// SIMATIC S7-200 project (STEP 7-Micro/WIN), CPU 226 REL 02.00

ORGANIZATION_BLOCK OB_1:OB1
TITLE=PROGRAM COMMENTS
BEGIN
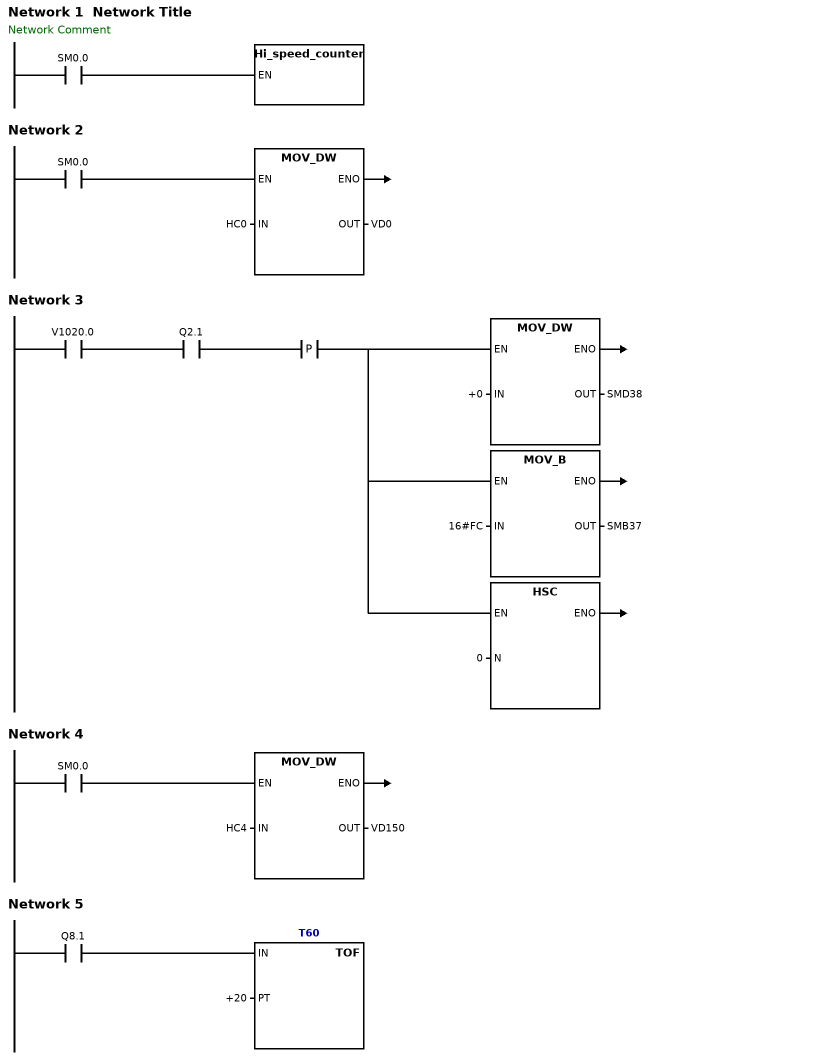
Network 1 // Network Title
// Network Comment
LD     SM0.0
CALL   Hi_speed_counter:SBR1
Network 2
LD     SM0.0
MOVD   HC0, VD0
Network 3
LD     V1020.0
A      Q2.1
EU
MOVD   +0, SMD38
MOVB   16#FC, SMB37
HSC    0
Network 4
LD     SM0.0
MOVD   HC4, VD150
Network 5
LD     Q8.1
TOF    T60, +20
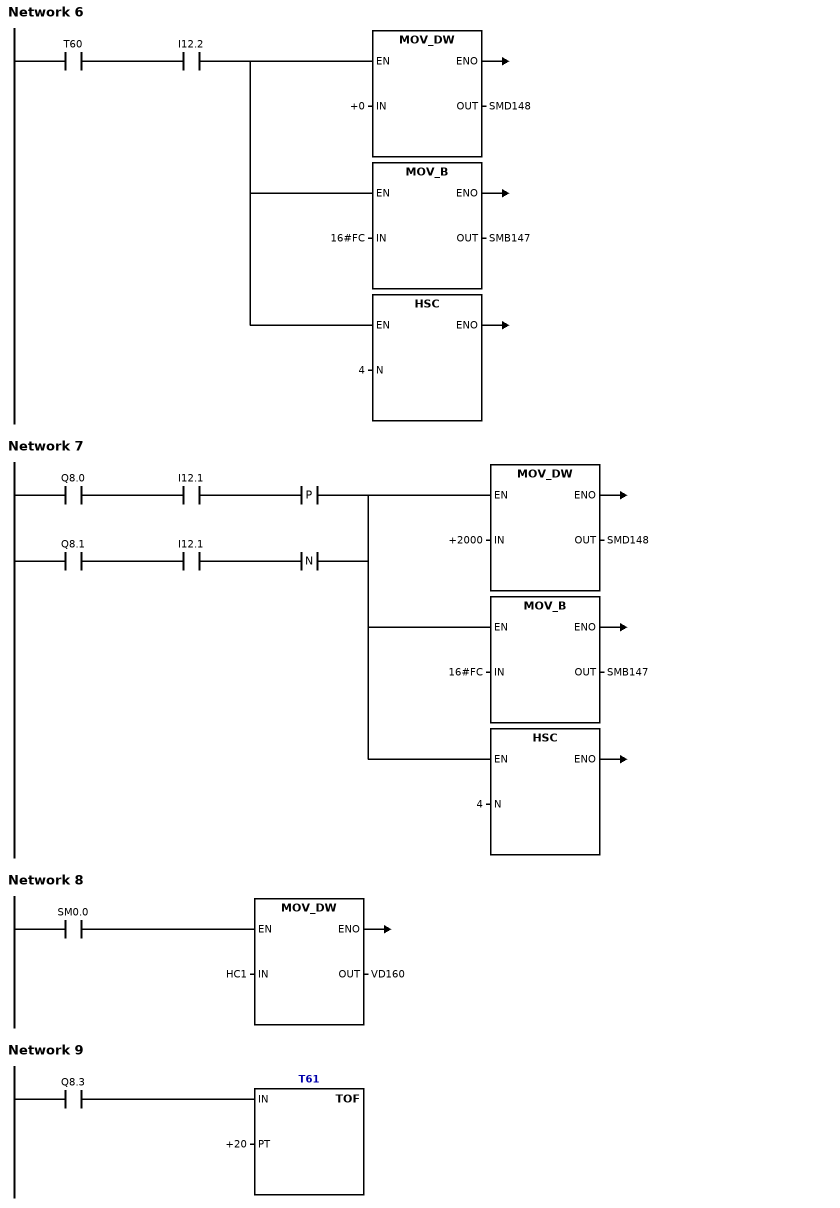
Network 6
LD     T60
A      I12.2
MOVD   +0, SMD148
MOVB   16#FC, SMB147
HSC    4
Network 7
LD     Q8.0
A      I12.1
EU
LD     Q8.1
A      I12.1
ED
OLD
MOVD   +2000, SMD148
MOVB   16#FC, SMB147
HSC    4
Network 8
LD     SM0.0
MOVD   HC1, VD160
Network 9
LD     Q8.3
TOF    T61, +20
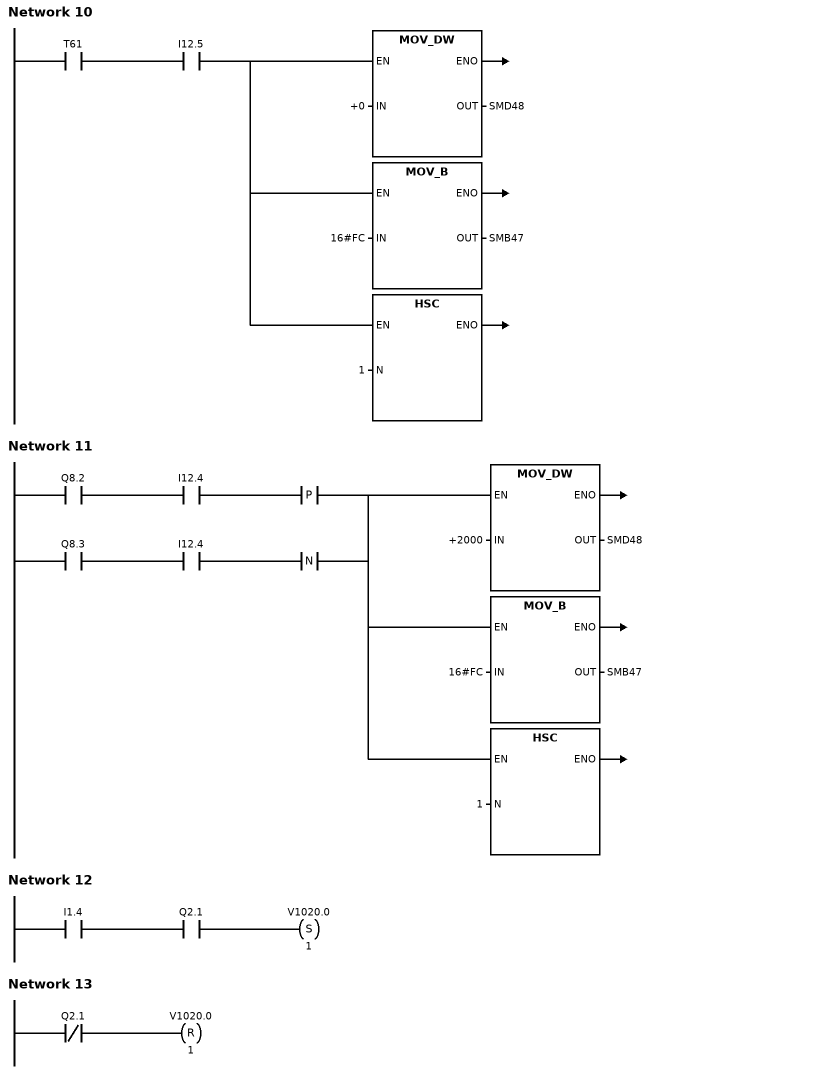
Network 10
LD     T61
A      I12.5
MOVD   +0, SMD48
MOVB   16#FC, SMB47
HSC    1
Network 11
LD     Q8.2
A      I12.4
EU
LD     Q8.3
A      I12.4
ED
OLD
MOVD   +2000, SMD48
MOVB   16#FC, SMB47
HSC    1
Network 12
LD     I1.4
A      Q2.1
S      V1020.0, 1
Network 13
LDN    Q2.1
R      V1020.0, 1
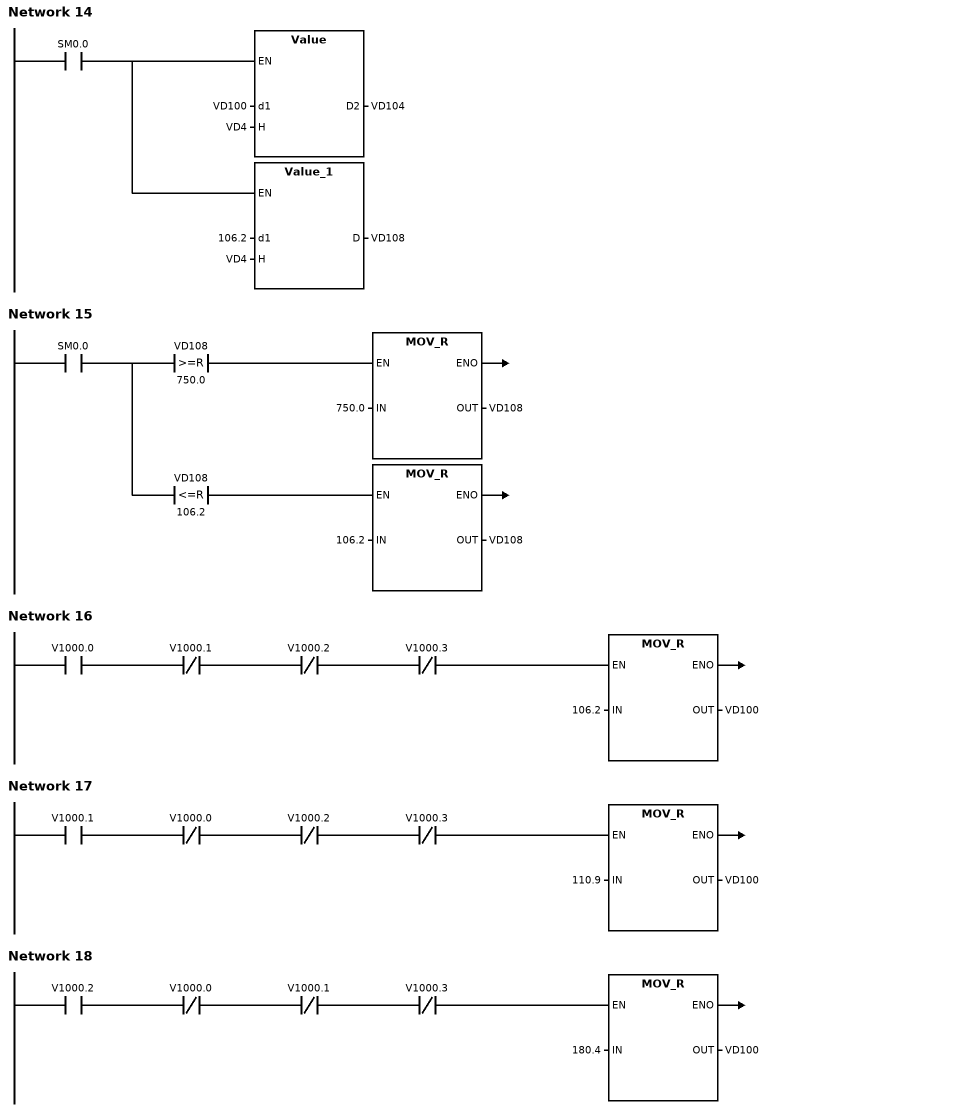
Network 14
LD     SM0.0
CALL   Value:SBR0, VD100, VD4, VD104
CALL   Value_1:SBR10, 106.2, VD4, VD108
Network 15
LD     SM0.0
LPS
AR>=   VD108, 750.0
MOVR   750.0, VD108
LPP
AR<=   VD108, 106.2
MOVR   106.2, VD108
Network 16
LD     V1000.0
AN     V1000.1
AN     V1000.2
AN     V1000.3
MOVR   106.2, VD100
Network 17
LD     V1000.1
AN     V1000.0
AN     V1000.2
AN     V1000.3
MOVR   110.9, VD100
Network 18
LD     V1000.2
AN     V1000.0
AN     V1000.1
AN     V1000.3
MOVR   180.4, VD100
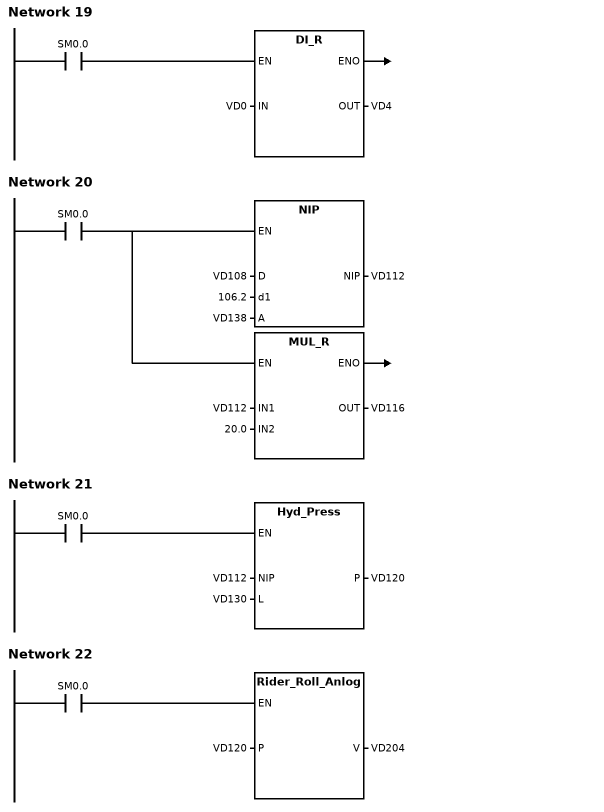
Network 19
LD     SM0.0
DTR    VD0, VD4
Network 20
LD     SM0.0
CALL   NIP:SBR2, VD108, 106.2, VD138, VD112
MOVR   VD112, VD116
*R     20.0, VD116
Network 21
LD     SM0.0
CALL   Hyd_Press:SBR3, VD112, VD130, VD120
Network 22
LD     SM0.0
CALL   Rider_Roll_Anlog:SBR4, VD120, VD204
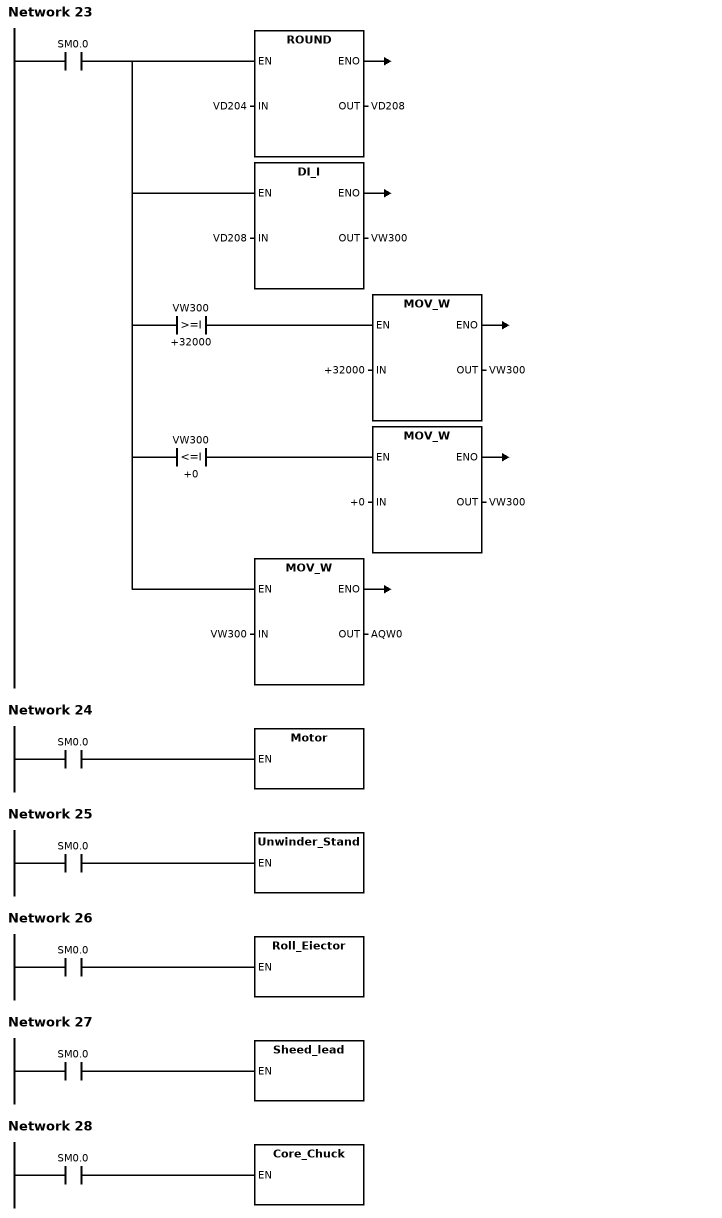
Network 23
LD     SM0.0
LPS
ROUND  VD204, VD208
DTI    VD208, VW300
AW>=   VW300, +32000
MOVW   +32000, VW300
LRD
AW<=   VW300, +0
MOVW   +0, VW300
LPP
MOVW   VW300, AQW0
Network 24
LD     SM0.0
CALL   Motor:SBR5
Network 25
LD     SM0.0
CALL   Unwinder_Stand:SBR6
Network 26
LD     SM0.0
CALL   Roll_Eiector:SBR7
Network 27
LD     SM0.0
CALL   Sheed_lead:SBR8
Network 28
LD     SM0.0
CALL   Core_Chuck:SBR9
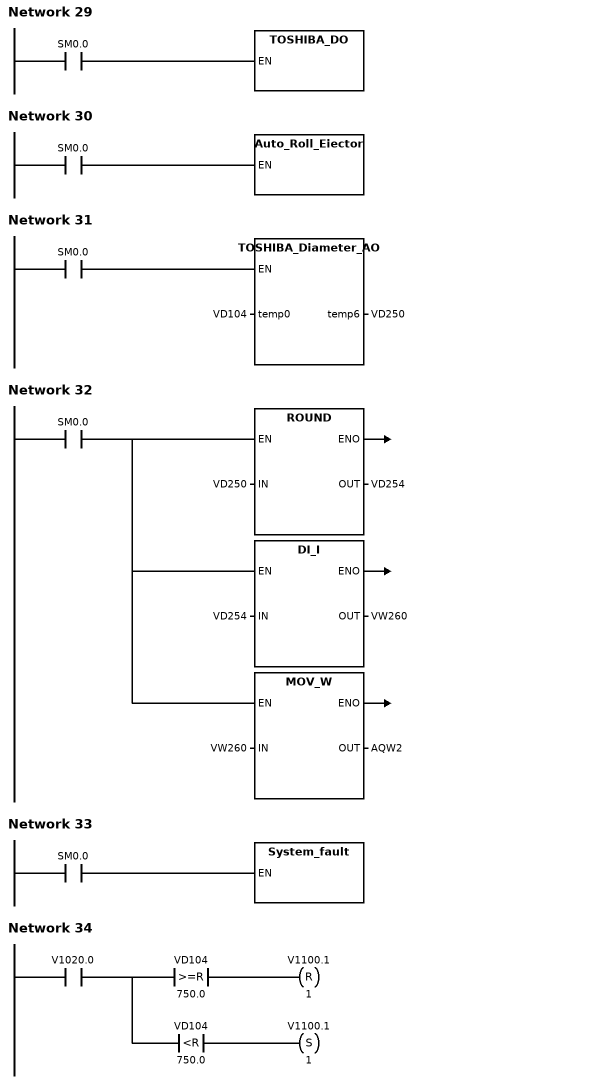
Network 29
LD     SM0.0
CALL   TOSHIBA_DO:SBR11
Network 30
LD     SM0.0
CALL   Auto_Roll_Eiector:SBR12
Network 31
LD     SM0.0
CALL   TOSHIBA_Diameter_AO:SBR13, VD104, VD250
Network 32
LD     SM0.0
ROUND  VD250, VD254
DTI    VD254, VW260
MOVW   VW260, AQW2
Network 33
LD     SM0.0
CALL   System_fault:SBR14
Network 34
LD     V1020.0
LPS
AR>=   VD104, 750.0
R      V1100.1, 1
LPP
AR<    VD104, 750.0
S      V1100.1, 1
END_ORGANIZATION_BLOCK

SUBROUTINE_BLOCK Value:SBR0
TITLE=SUBROUTINE COMMENTS
VAR_INPUT
d1:REAL;	// LD0 
H:REAL;	// LD4 
END_VAR
VAR_OUTPUT
D2:REAL;	// LD8 
END_VAR
BEGIN
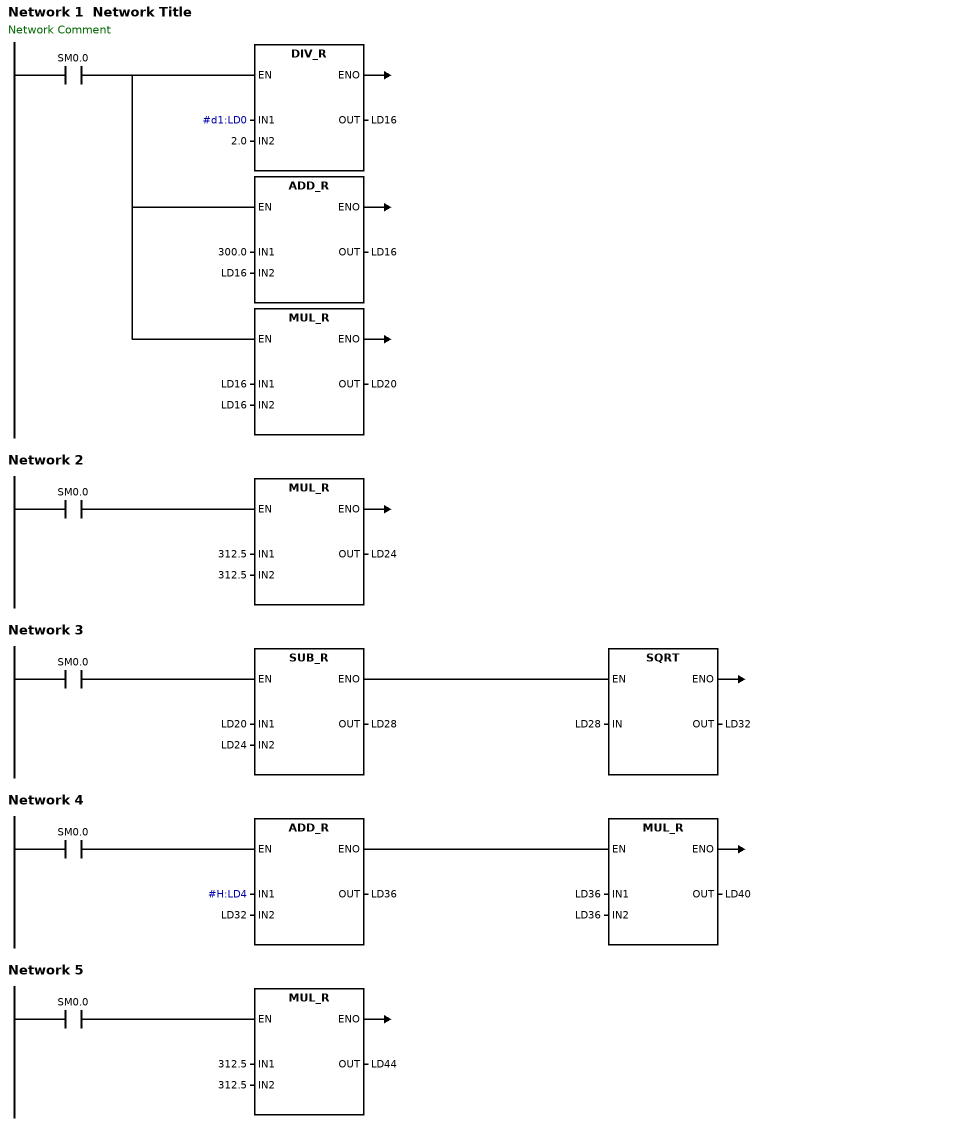
Network 1 // Network Title
// Network Comment
LD     SM0.0
MOVR   #d1:LD0, LD16
/R     2.0, LD16
+R     300.0, LD16
MOVR   LD16, LD20
*R     LD16, LD20
Network 2
LD     SM0.0
MOVR   312.5, LD24
*R     312.5, LD24
Network 3
LD     SM0.0
MOVR   LD20, LD28
AENO
-R     LD24, LD28
AENO
SQRT   LD28, LD32
Network 4
LD     SM0.0
MOVR   #H:LD4, LD36
AENO
+R     LD32, LD36
AENO
MOVR   LD36, LD40
*R     LD36, LD40
Network 5
LD     SM0.0
MOVR   312.5, LD44
*R     312.5, LD44
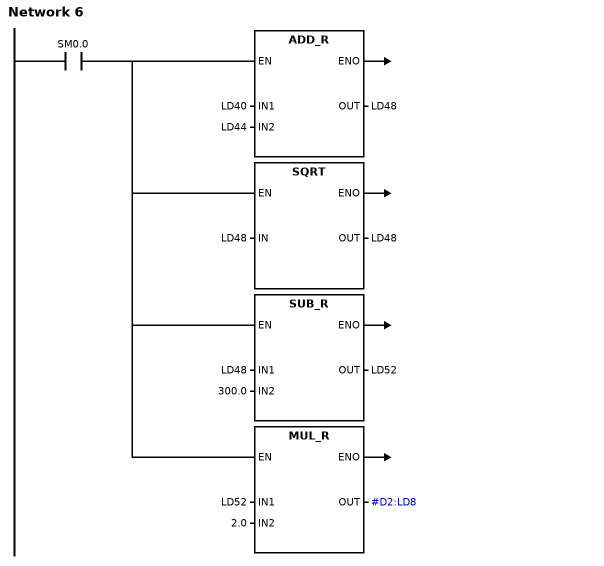
Network 6
LD     SM0.0
MOVR   LD40, LD48
+R     LD44, LD48
SQRT   LD48, LD48
MOVR   LD48, LD52
-R     300.0, LD52
MOVR   LD52, #D2:LD8
*R     2.0, #D2:LD8
END_SUBROUTINE_BLOCK

SUBROUTINE_BLOCK Hi_speed_counter:SBR1
TITLE=
BEGIN
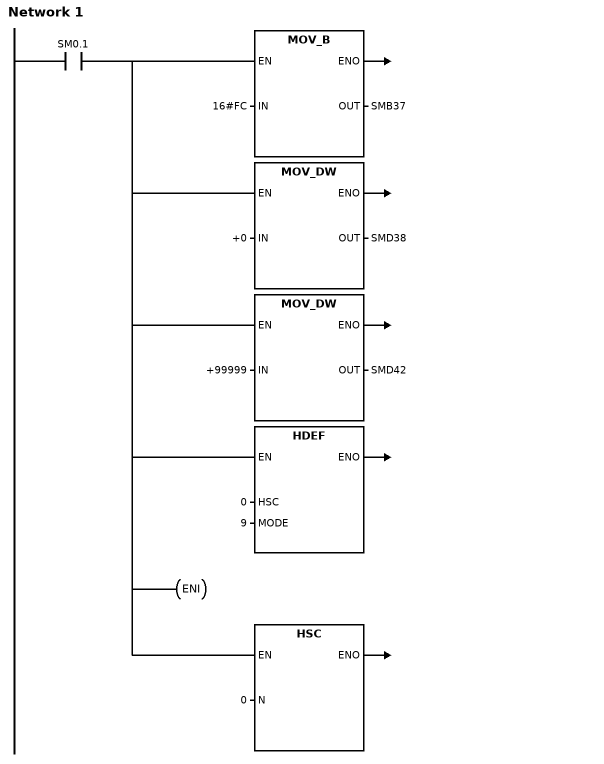
Network 1
LD     SM0.1
MOVB   16#FC, SMB37
MOVD   +0, SMD38
MOVD   +99999, SMD42
HDEF   0, 9
ENI
HSC    0
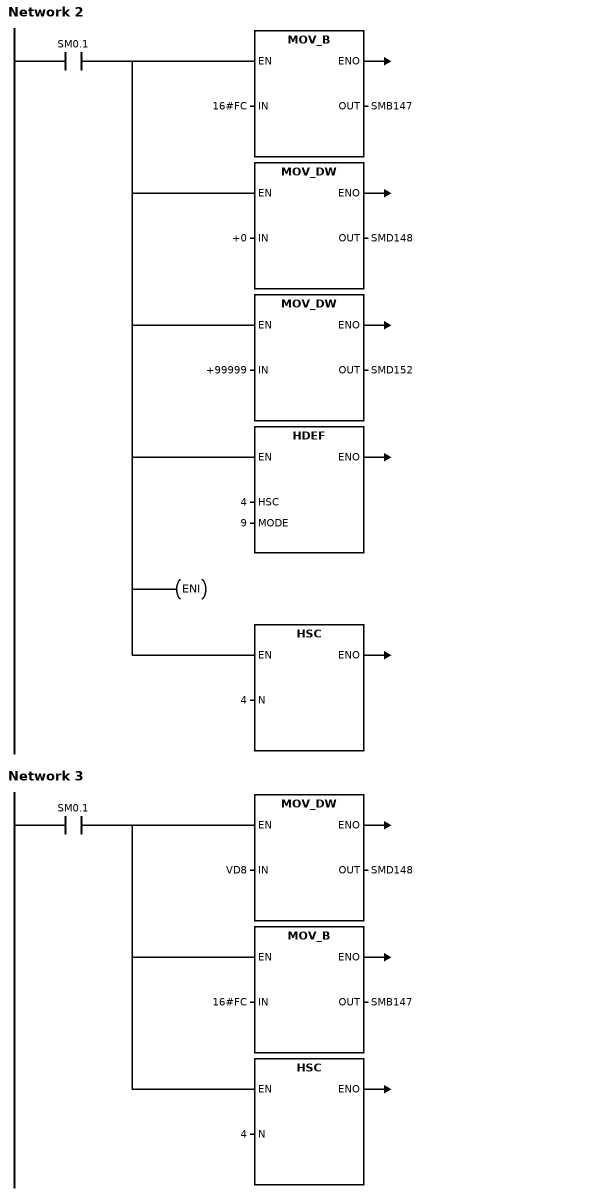
Network 2
LD     SM0.1
MOVB   16#FC, SMB147
MOVD   +0, SMD148
MOVD   +99999, SMD152
HDEF   4, 9
ENI
HSC    4
Network 3
LD     SM0.1
MOVD   VD8, SMD148
MOVB   16#FC, SMB147
HSC    4
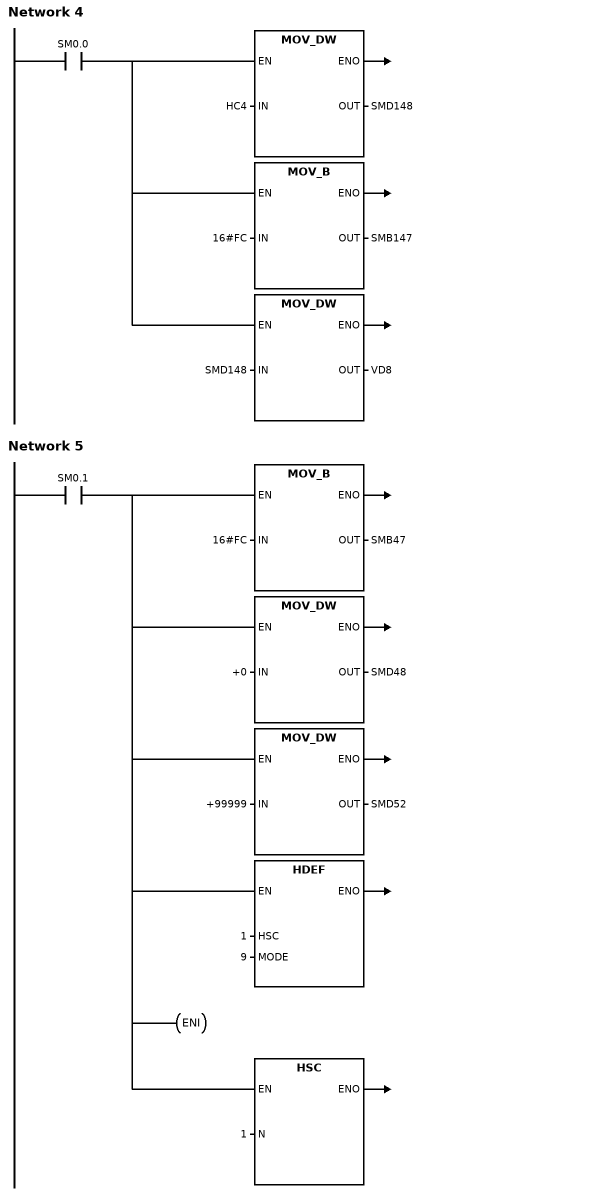
Network 4
LD     SM0.0
MOVD   HC4, SMD148
MOVB   16#FC, SMB147
MOVD   SMD148, VD8
Network 5
LD     SM0.1
MOVB   16#FC, SMB47
MOVD   +0, SMD48
MOVD   +99999, SMD52
HDEF   1, 9
ENI
HSC    1
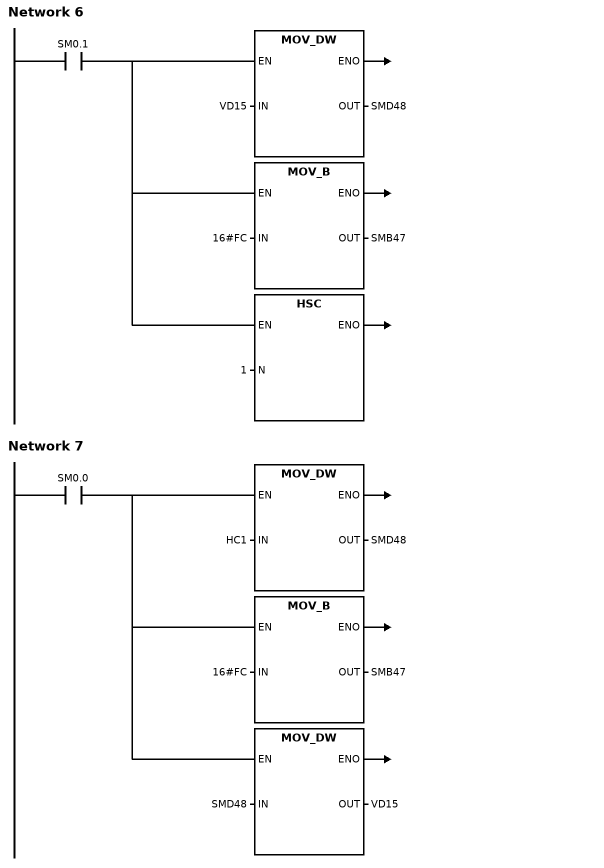
Network 6
LD     SM0.1
MOVD   VD15, SMD48
MOVB   16#FC, SMB47
HSC    1
Network 7
LD     SM0.0
MOVD   HC1, SMD48
MOVB   16#FC, SMB47
MOVD   SMD48, VD15
END_SUBROUTINE_BLOCK

SUBROUTINE_BLOCK NIP:SBR2
TITLE=
VAR_INPUT
D:REAL;	// LD0 
d1:REAL;	// LD4 
A:REAL;	// LD8 
END_VAR
VAR_OUTPUT
NIP:REAL;	// LD12 
END_VAR
BEGIN
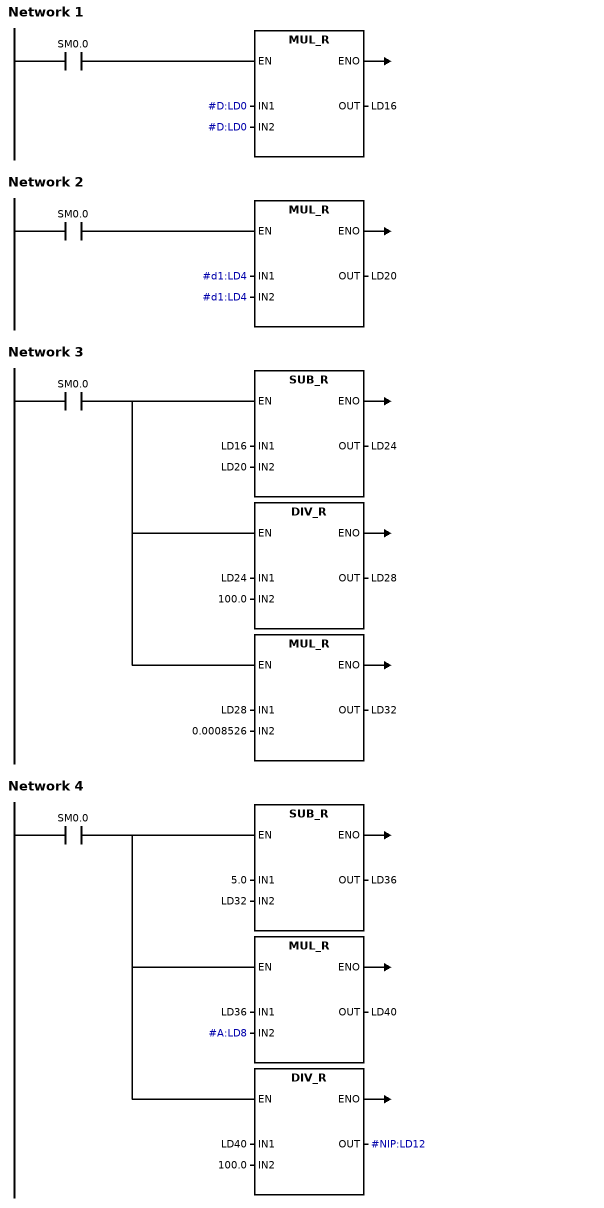
Network 1
LD     SM0.0
MOVR   #D:LD0, LD16
*R     #D:LD0, LD16
Network 2
LD     SM0.0
MOVR   #d1:LD4, LD20
*R     #d1:LD4, LD20
Network 3
LD     SM0.0
MOVR   LD16, LD24
-R     LD20, LD24
MOVR   LD24, LD28
/R     100.0, LD28
MOVR   LD28, LD32
*R     0.0008526, LD32
Network 4
LD     SM0.0
MOVR   5.0, LD36
-R     LD32, LD36
MOVR   LD36, LD40
*R     #A:LD8, LD40
MOVR   LD40, #NIP:LD12
/R     100.0, #NIP:LD12
END_SUBROUTINE_BLOCK

SUBROUTINE_BLOCK Hyd_Press:SBR3
TITLE=
VAR_INPUT
NIP:REAL;	// LD0 
L:REAL;	// LD4 
END_VAR
VAR_OUTPUT
P:REAL;	// LD8 
END_VAR
BEGIN
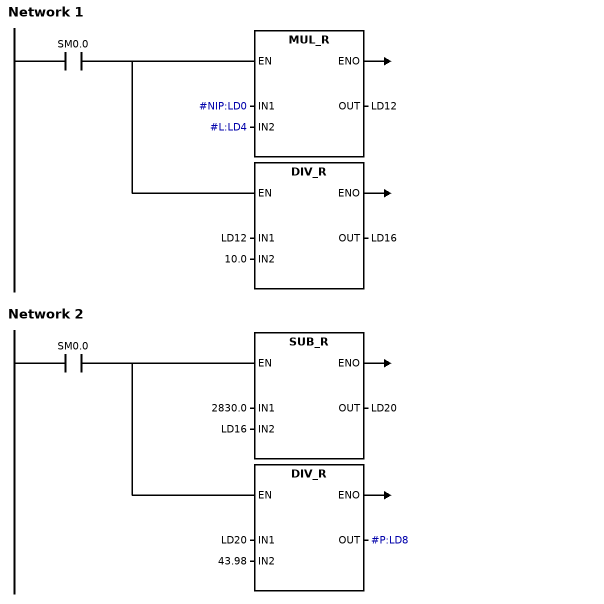
Network 1
LD     SM0.0
MOVR   #NIP:LD0, LD12
*R     #L:LD4, LD12
MOVR   LD12, LD16
/R     10.0, LD16
Network 2
LD     SM0.0
MOVR   2830.0, LD20
-R     LD16, LD20
MOVR   LD20, #P:LD8
/R     43.98, #P:LD8
END_SUBROUTINE_BLOCK

SUBROUTINE_BLOCK Rider_Roll_Anlog:SBR4
TITLE=
VAR_INPUT
P:REAL;	// LD0 
END_VAR
VAR_OUTPUT
V:REAL;	// LD4 
END_VAR
BEGIN
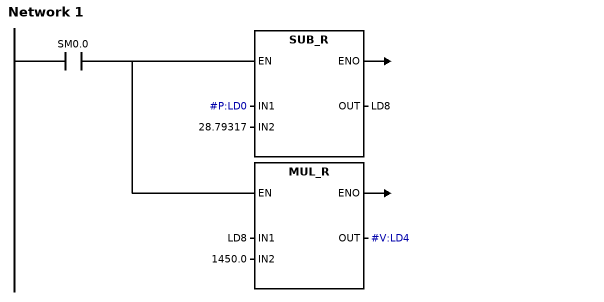
Network 1
LD     SM0.0
MOVR   #P:LD0, LD8
-R     28.79317, LD8
MOVR   LD8, #V:LD4
*R     1450.0, #V:LD4
END_SUBROUTINE_BLOCK

SUBROUTINE_BLOCK Motor:SBR5
TITLE=
BEGIN
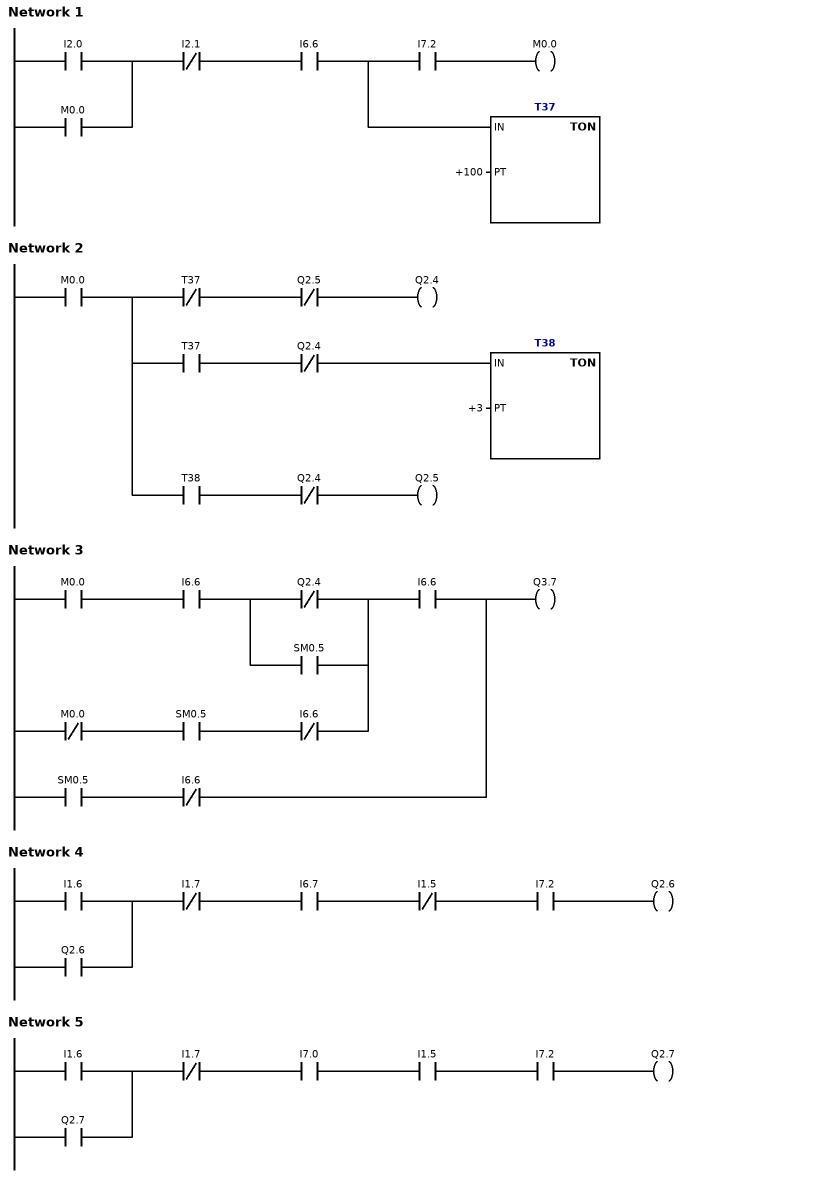
Network 1
LD     I2.0
O      M0.0
AN     I2.1
A      I6.6
LPS
A      I7.2
=      M0.0
LPP
TON    T37, +100
Network 2
LD     M0.0
LPS
AN     T37
AN     Q2.5
=      Q2.4
LRD
A      T37
AN     Q2.4
TON    T38, +3
LPP
A      T38
AN     Q2.4
=      Q2.5
Network 3
LD     M0.0
A      I6.6
LDN    Q2.4
O      SM0.5
ALD
LDN    M0.0
A      SM0.5
AN     I6.6
OLD
A      I6.6
LD     SM0.5
AN     I6.6
OLD
=      Q3.7
Network 4
LD     I1.6
O      Q2.6
AN     I1.7
A      I6.7
AN     I1.5
A      I7.2
=      Q2.6
Network 5
LD     I1.6
O      Q2.7
AN     I1.7
A      I7.0
A      I1.5
A      I7.2
=      Q2.7
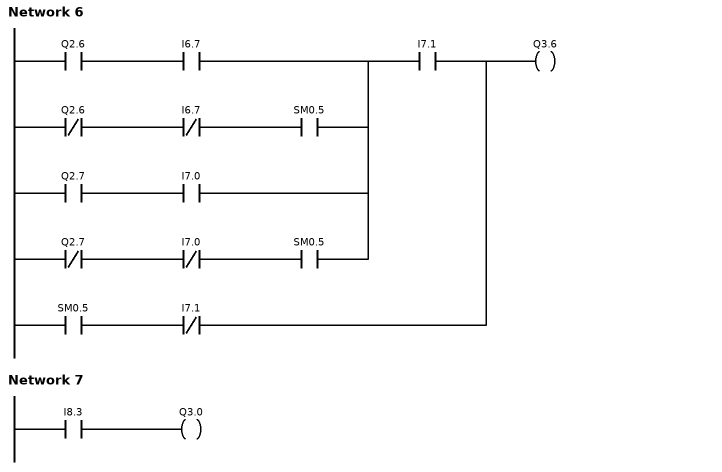
Network 6
LD     Q2.6
A      I6.7
LDN    Q2.6
AN     I6.7
A      SM0.5
OLD
LD     Q2.7
A      I7.0
OLD
LDN    Q2.7
AN     I7.0
A      SM0.5
OLD
A      I7.1
LD     SM0.5
AN     I7.1
OLD
=      Q3.6
Network 7
LD     I8.3
=      Q3.0
END_SUBROUTINE_BLOCK

SUBROUTINE_BLOCK Unwinder_Stand:SBR6
TITLE=
BEGIN
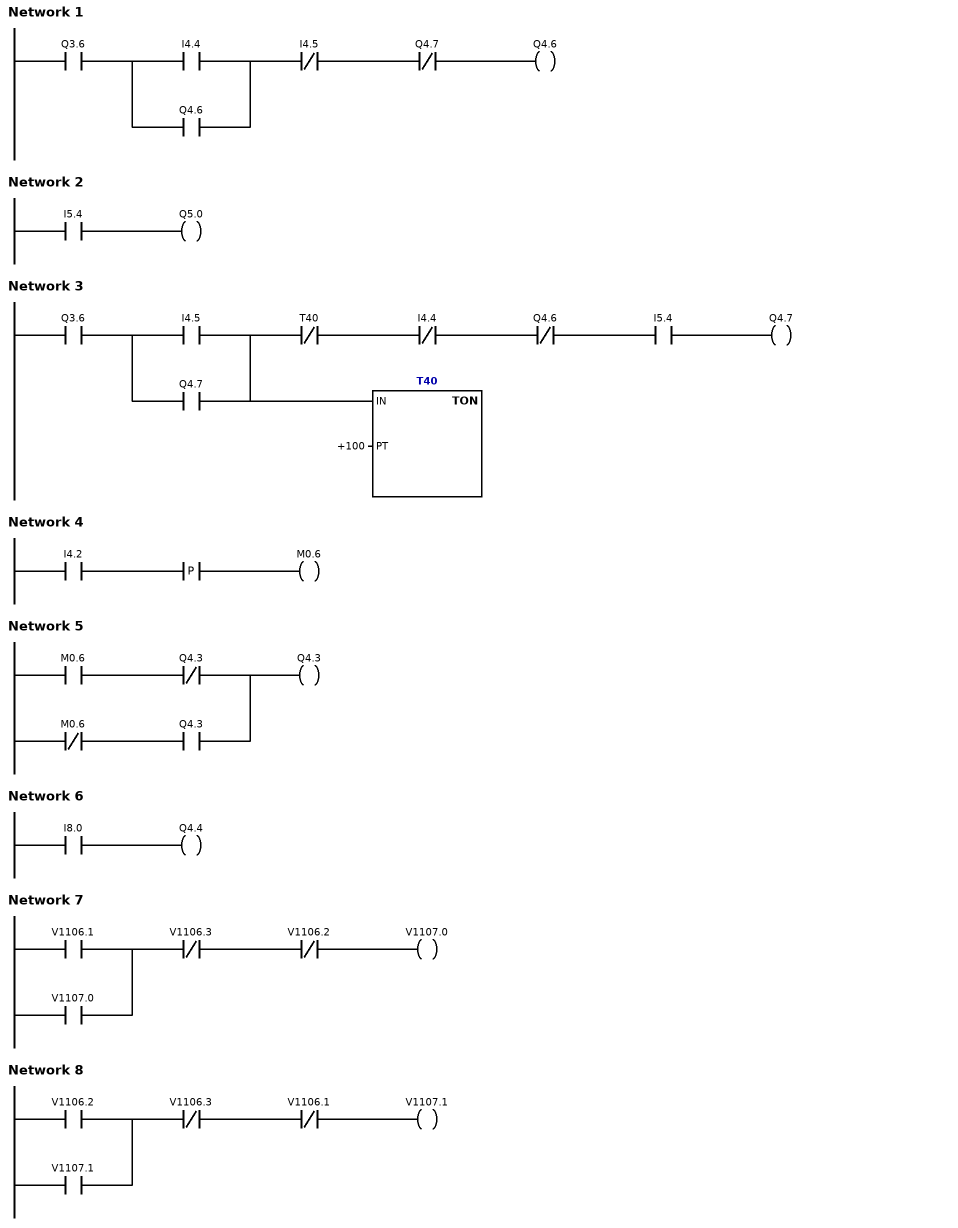
Network 1
LD     Q3.6
LD     I4.4
O      Q4.6
ALD
AN     I4.5
AN     Q4.7
=      Q4.6
Network 2
LD     I5.4
=      Q5.0
Network 3
LD     Q3.6
LD     I4.5
O      Q4.7
ALD
LPS
AN     T40
AN     I4.4
AN     Q4.6
A      I5.4
=      Q4.7
LPP
TON    T40, +100
Network 4
LD     I4.2
EU
=      M0.6
Network 5
LD     M0.6
AN     Q4.3
LDN    M0.6
A      Q4.3
OLD
=      Q4.3
Network 6
LD     I8.0
=      Q4.4
Network 7
LD     V1106.1
O      V1107.0
AN     V1106.3
AN     V1106.2
=      V1107.0
Network 8
LD     V1106.2
O      V1107.1
AN     V1106.3
AN     V1106.1
=      V1107.1
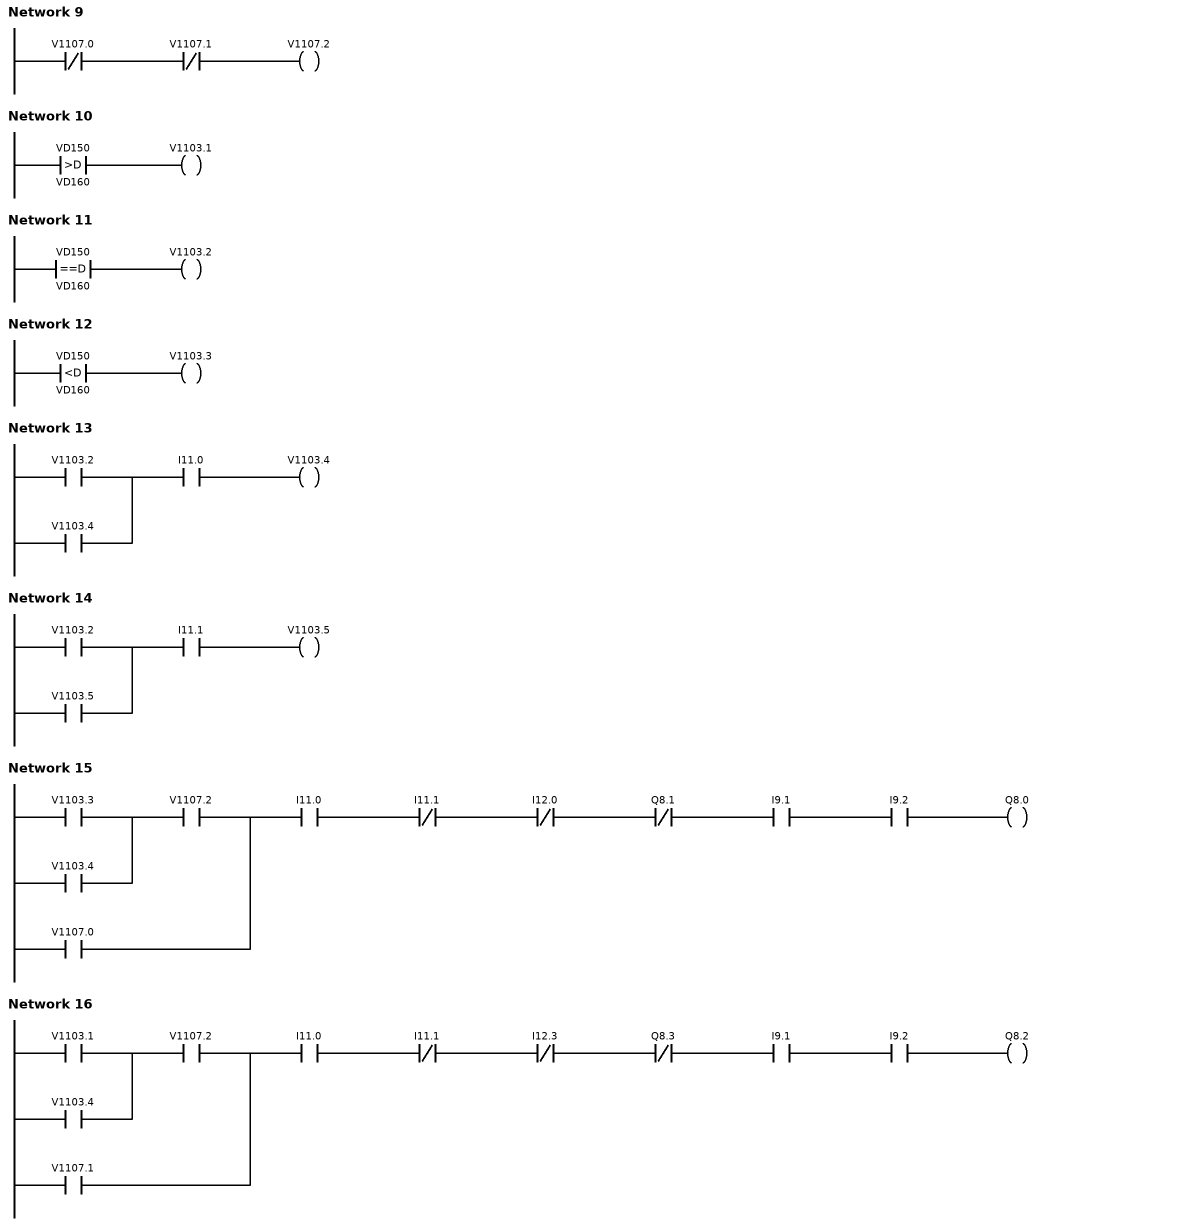
Network 9
LDN    V1107.0
AN     V1107.1
=      V1107.2
Network 10
LDD>   VD150, VD160
=      V1103.1
Network 11
LDD=   VD150, VD160
=      V1103.2
Network 12
LDD<   VD150, VD160
=      V1103.3
Network 13
LD     V1103.2
O      V1103.4
A      I11.0
=      V1103.4
Network 14
LD     V1103.2
O      V1103.5
A      I11.1
=      V1103.5
Network 15
LD     V1103.3
O      V1103.4
A      V1107.2
O      V1107.0
A      I11.0
AN     I11.1
AN     I12.0
AN     Q8.1
A      I9.1
A      I9.2
=      Q8.0
Network 16
LD     V1103.1
O      V1103.4
A      V1107.2
O      V1107.1
A      I11.0
AN     I11.1
AN     I12.3
AN     Q8.3
A      I9.1
A      I9.2
=      Q8.2
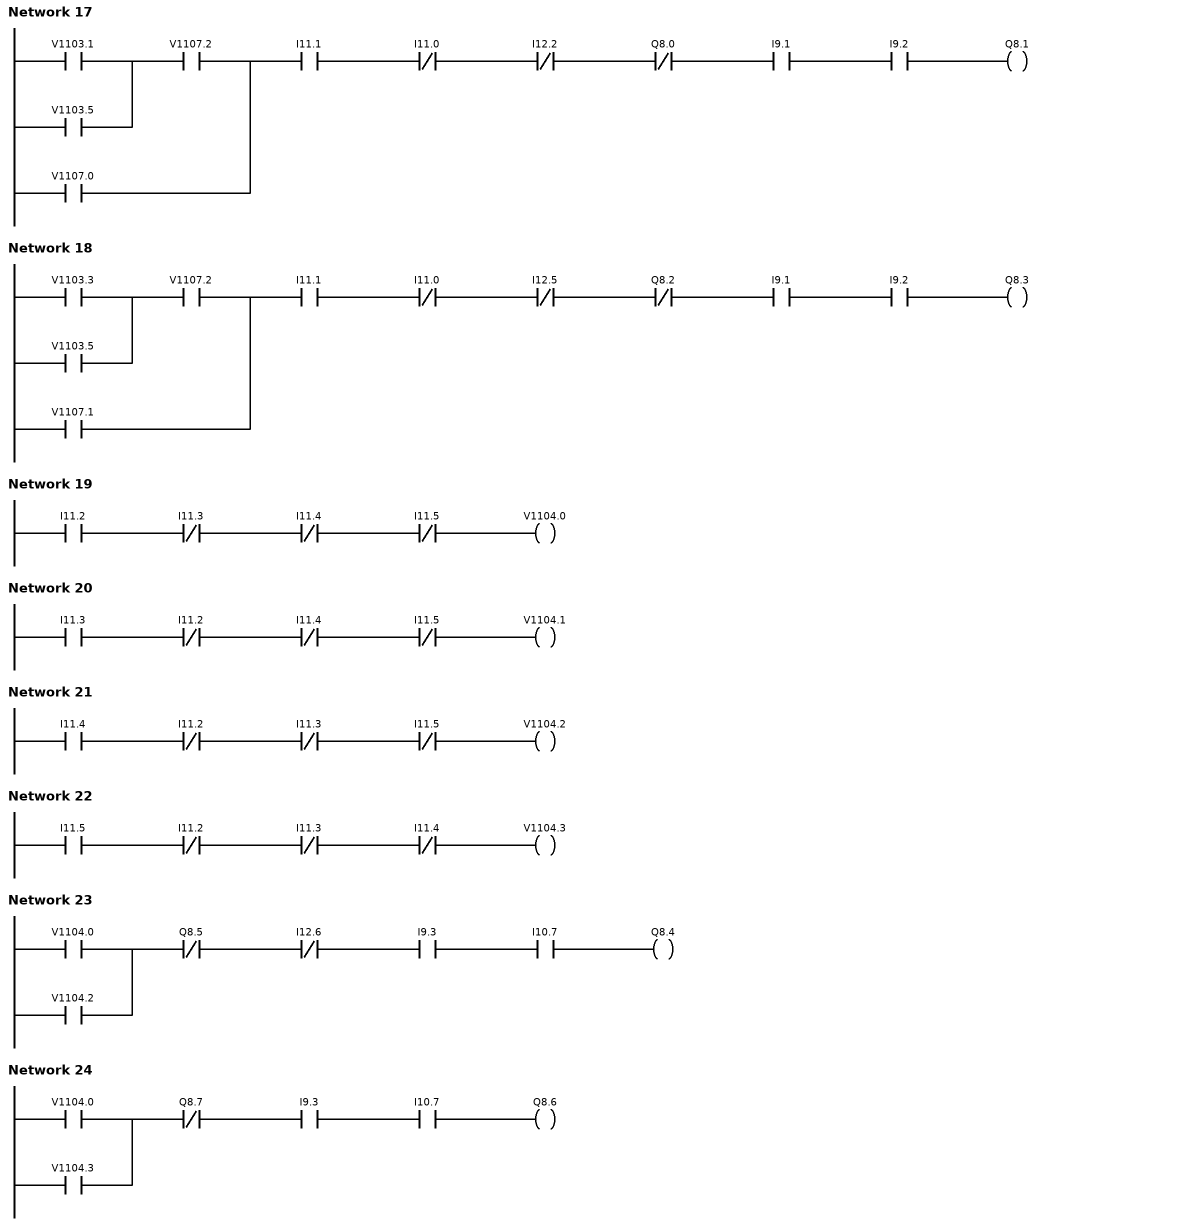
Network 17
LD     V1103.1
O      V1103.5
A      V1107.2
O      V1107.0
A      I11.1
AN     I11.0
AN     I12.2
AN     Q8.0
A      I9.1
A      I9.2
=      Q8.1
Network 18
LD     V1103.3
O      V1103.5
A      V1107.2
O      V1107.1
A      I11.1
AN     I11.0
AN     I12.5
AN     Q8.2
A      I9.1
A      I9.2
=      Q8.3
Network 19
LD     I11.2
AN     I11.3
AN     I11.4
AN     I11.5
=      V1104.0
Network 20
LD     I11.3
AN     I11.2
AN     I11.4
AN     I11.5
=      V1104.1
Network 21
LD     I11.4
AN     I11.2
AN     I11.3
AN     I11.5
=      V1104.2
Network 22
LD     I11.5
AN     I11.2
AN     I11.3
AN     I11.4
=      V1104.3
Network 23
LD     V1104.0
O      V1104.2
AN     Q8.5
AN     I12.6
A      I9.3
A      I10.7
=      Q8.4
Network 24
LD     V1104.0
O      V1104.3
AN     Q8.7
A      I9.3
A      I10.7
=      Q8.6
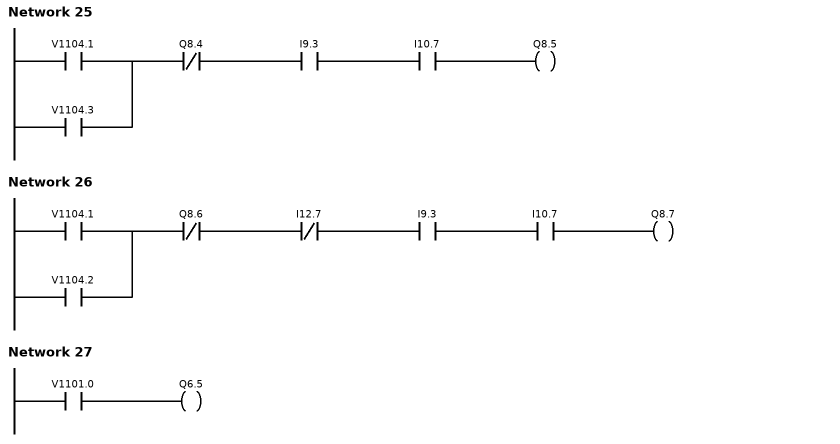
Network 25
LD     V1104.1
O      V1104.3
AN     Q8.4
A      I9.3
A      I10.7
=      Q8.5
Network 26
LD     V1104.1
O      V1104.2
AN     Q8.6
AN     I12.7
A      I9.3
A      I10.7
=      Q8.7
Network 27
LD     V1101.0
=      Q6.5
END_SUBROUTINE_BLOCK

SUBROUTINE_BLOCK Roll_Eiector:SBR7
TITLE=
BEGIN
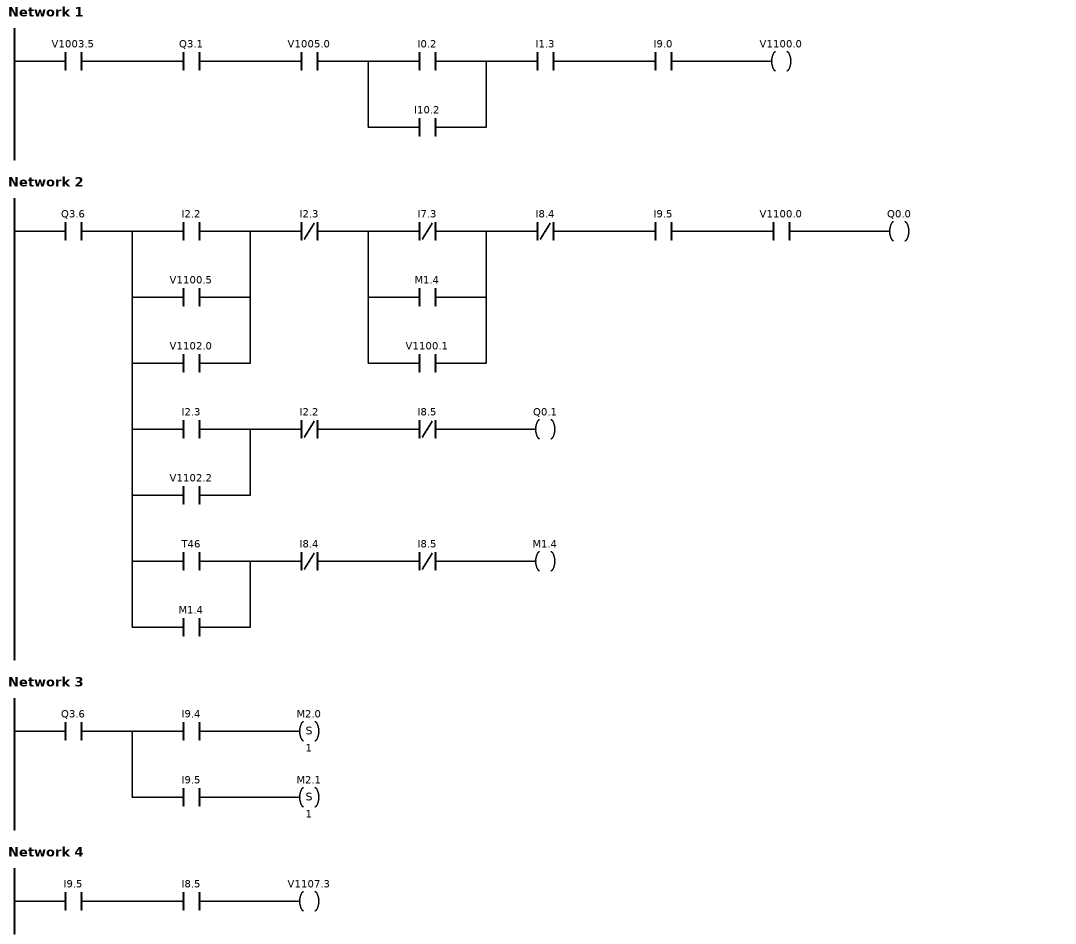
Network 1
LD     V1003.5
A      Q3.1
A      V1005.0
LD     I0.2
O      I10.2
ALD
A      I1.3
A      I9.0
=      V1100.0
Network 2
LD     Q3.6
LPS
LD     I2.2
O      V1100.5
O      V1102.0
AN     I2.3
LDN    I7.3
O      M1.4
O      V1100.1
ALD
ALD
AN     I8.4
A      I9.5
A      V1100.0
=      Q0.0
LRD
LD     I2.3
O      V1102.2
ALD
AN     I2.2
AN     I8.5
=      Q0.1
LPP
LD     T46
O      M1.4
ALD
AN     I8.4
AN     I8.5
=      M1.4
Network 3
LD     Q3.6
LPS
A      I9.4
S      M2.0, 1
LPP
A      I9.5
S      M2.1, 1
Network 4
LD     I9.5
A      I8.5
=      V1107.3
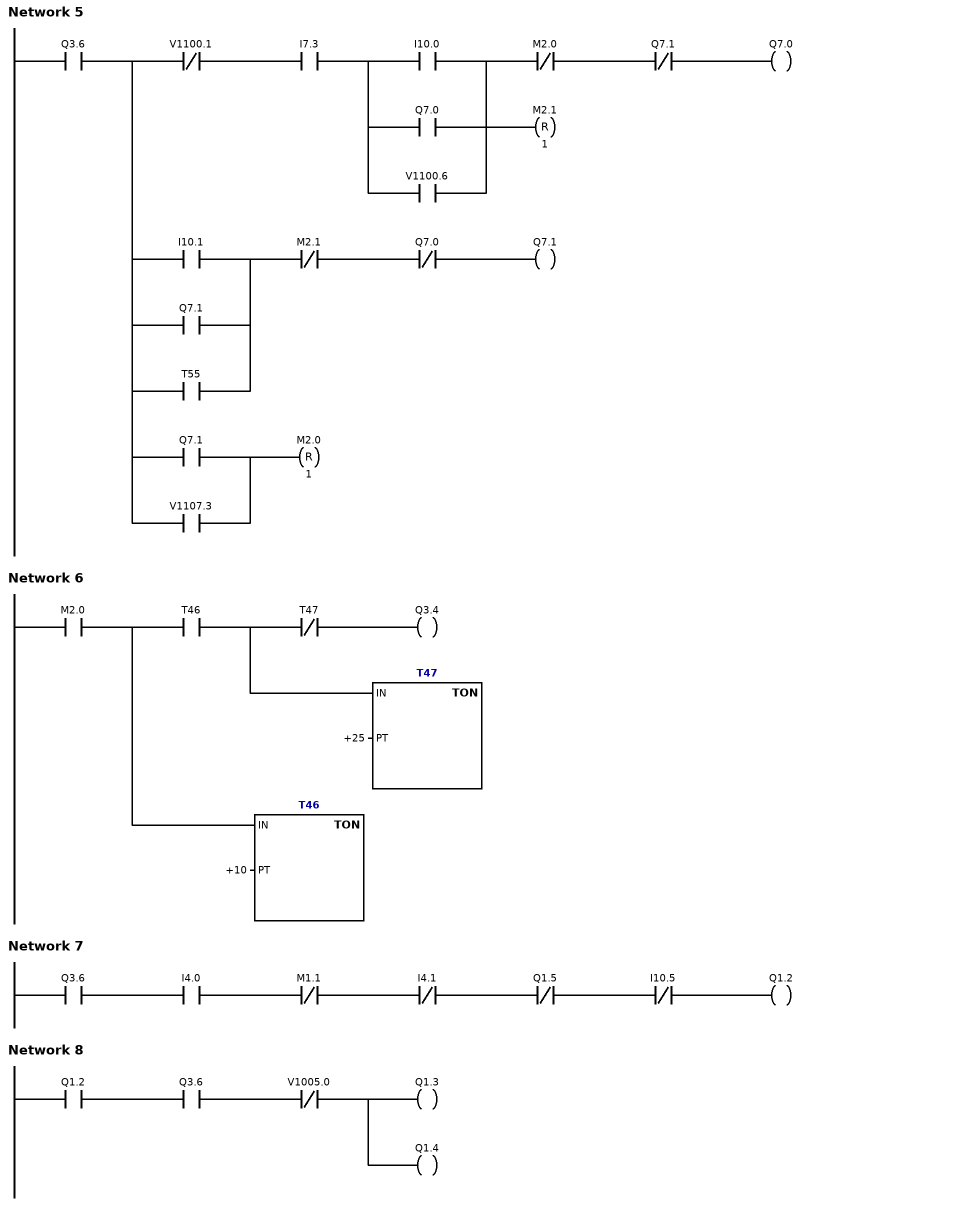
Network 5
LD     Q3.6
LPS
AN     V1100.1
A      I7.3
LD     I10.0
O      Q7.0
O      V1100.6
ALD
LPS
AN     M2.0
AN     Q7.1
=      Q7.0
LPP
R      M2.1, 1
LRD
LD     I10.1
O      Q7.1
O      T55
ALD
AN     M2.1
AN     Q7.0
=      Q7.1
LPP
LD     Q7.1
O      V1107.3
ALD
R      M2.0, 1
Network 6
LD     M2.0
LPS
A      T46
LPS
AN     T47
=      Q3.4
LPP
TON    T47, +25
LPP
TON    T46, +10
Network 7
LD     Q3.6
A      I4.0
AN     M1.1
AN     I4.1
AN     Q1.5
AN     I10.5
=      Q1.2
Network 8
LD     Q1.2
A      Q3.6
AN     V1005.0
=      Q1.3
=      Q1.4
